{attribute 'GeneratedUsingTerminal: EL2032-0000-0018'}
{attribute addProperty BoxType "EL2032-0000-0018"}
{attribute addProperty Id "EtcSlaveTerminalBaseDiag_1AT %I*Diag_A72B1E171Diag_2AT %I*Diag_A72B1E171Channel_1AT %Q*Channel_42CA91F71Channel_2AT %Q*Channel_42CA91F71WcStateAT %I*WcState_9091E0EB2InfoDataAT %I*InfoData_6F19DB2B2"}
{attribute addProperty CRC "3094279553"}
{attribute addProperty Size "8"}
TYPE EL2032_B86EF581 EXTENDS EtcSlaveTerminalBase :
STRUCT
	{attribute addProperty Name "Diag_1"}
	Diag_1 : Diag_A72B1E17;
	{attribute addProperty Name "Diag_2"}
	Diag_2 : Diag_A72B1E17;
	{attribute addProperty Name "Channel_1"}
	Channel_1 : Channel_42CA91F7;
	{attribute addProperty Name "Channel_2"}
	Channel_2 : Channel_42CA91F7;
	{attribute addProperty Name "WcState"}
	WcState : WcState_9091E0EB;
	{attribute addProperty Name "InfoData"}
	InfoData : InfoData_6F19DB2B;
END_STRUCT
END_TYPE

(* stored: Version 1.2.0.0, ProductVersion 3.1.4024.9
   DUT EL2032_B86EF581: Id {ff8c141d-253a-4404-ad77-7183bc4bf63b} *)
